{attribute 'qualified_only'}
{attribute 'strict'}
TYPE E_CRYO_CRYOTELGT_CMD :
(
	NONE := 0,
	OFF,
	ON,
	SET_POWER
);
END_TYPE

(* stored: Version 1.1.0.1, ProductVersion 3.1.4024.12
   DUT E_CRYO_CRYOTELGT_CMD: Id {2ad4b6e0-e58c-4389-942b-50fe3ff1499e} *)
